Staubli VAL3: clkAllOn.pgx

program clkAllOn()
  local num index
begin
  for index=0 to 31
    if statusValves[index]==0
      call toggleValve(index)
    endIf
  endFor

end
